// TIA Portal V20 export
FUNCTION_BLOCK "Sequence_1_SepaUnwinderTop"   // FB202, LAD
AUTHOR : ERsystem_FA2_DH. Kim
// stored: IsIECCheckEnabled true, MemoryReserve 100, Namespace Unit1.Em0, SetENOAutomatically false
   VAR
      statSelectedJobNumber { ExternalWritable := 'False'} : DInt;   // Evaluated Job Number
      instSequenceLADStatus { ExternalWritable := 'False'} : "LAF_StatusLadSequence";
      instSequenceLADControl { ExternalWritable := 'False'} : "LAF_ControlLadSequence";
      statTonTime { ExternalAccessible := 'False'; ExternalVisible := 'False'; ExternalWritable := 'False'} : Array[0..1999] of TON_TIME;
   END_VAR
   VAR CONSTANT
      STEP_IDLE : DInt := 1;
      STEP_IMMEDIATE_STOP : DInt := 9001;   // Step executed when an immediate stop command is triggered for the sequence (i.e. when unit is in state aborting)
      JOB_1_STEP_01 : DInt := 101;
      JOB_1_STEP_10 : DInt := 110;
      JOB_1_STEP_20 : DInt := 120;
      JOB_1_STEP_80 : DInt := 180;
      JOB_1_STEP_81 : DInt := 181;
      JOB_1_STEP_90 : DInt := 190;
      JOB_2_STEP_01 : DInt := 201;
      JOB_2_STEP_80 : DInt := 280;
      JOB_2_STEP_90 : DInt := 290;
      JOB_10_STEP_01 : DInt := 1001;
      JOB_10_STEP_80 : DInt := 1080;
      JOB_10_STEP_90 : DInt := 1090;
      FALSE : Bool := FALSE;
      TRUE : Bool := TRUE;
   END_VAR
   VAR_TEMP   // added for the SCL form of the ladder/FBD networks
      _w1 : Bool;
      _w2 : Bool;
   END_VAR
BEGIN

REGION Network 1: BLOCK INFO HEADER
   // (company) / (C) Copyright (year)
   // ---------------------------------------------------------------------------------
   // Title:                             (Title of this block)
   // Comment/Function: (that is implemented in the block)
   // Library/Family:           (that the source is dedicated to)
   // Author:                        (department / person in charge / contact)
   // Target System:          (test system with FW version)
   // Engineering:              TIA Portal (SW version)
   // Restrictions:               (OB types, etc.)
   // Requirements:           (hardware, technological package, etc.)
   // ---------------------------------------------------------------------------------
   // Change log table:
   // Version          | Date             | Signature      | Expert in charge  | Changes applied ------------------------|----------------------|-------------------------|--------------------------------|-----------------------
   // 001.000.000 | yyyy-mm-dd | 0x00000000 | (name of expert) | First released version
END_REGION

REGION Network 2: DESCRIPTION
   // This is a template block provided by the Automation Framework. It can be used to create an own project.
   // The Block Info Header is prepared to put in your own data.
   // Description of the block could be added here and the docu created by Code2Docu.
END_REGION

REGION Network 3: ********************* CONTROL *************************
END_REGION

REGION Network 4: Sequence Control
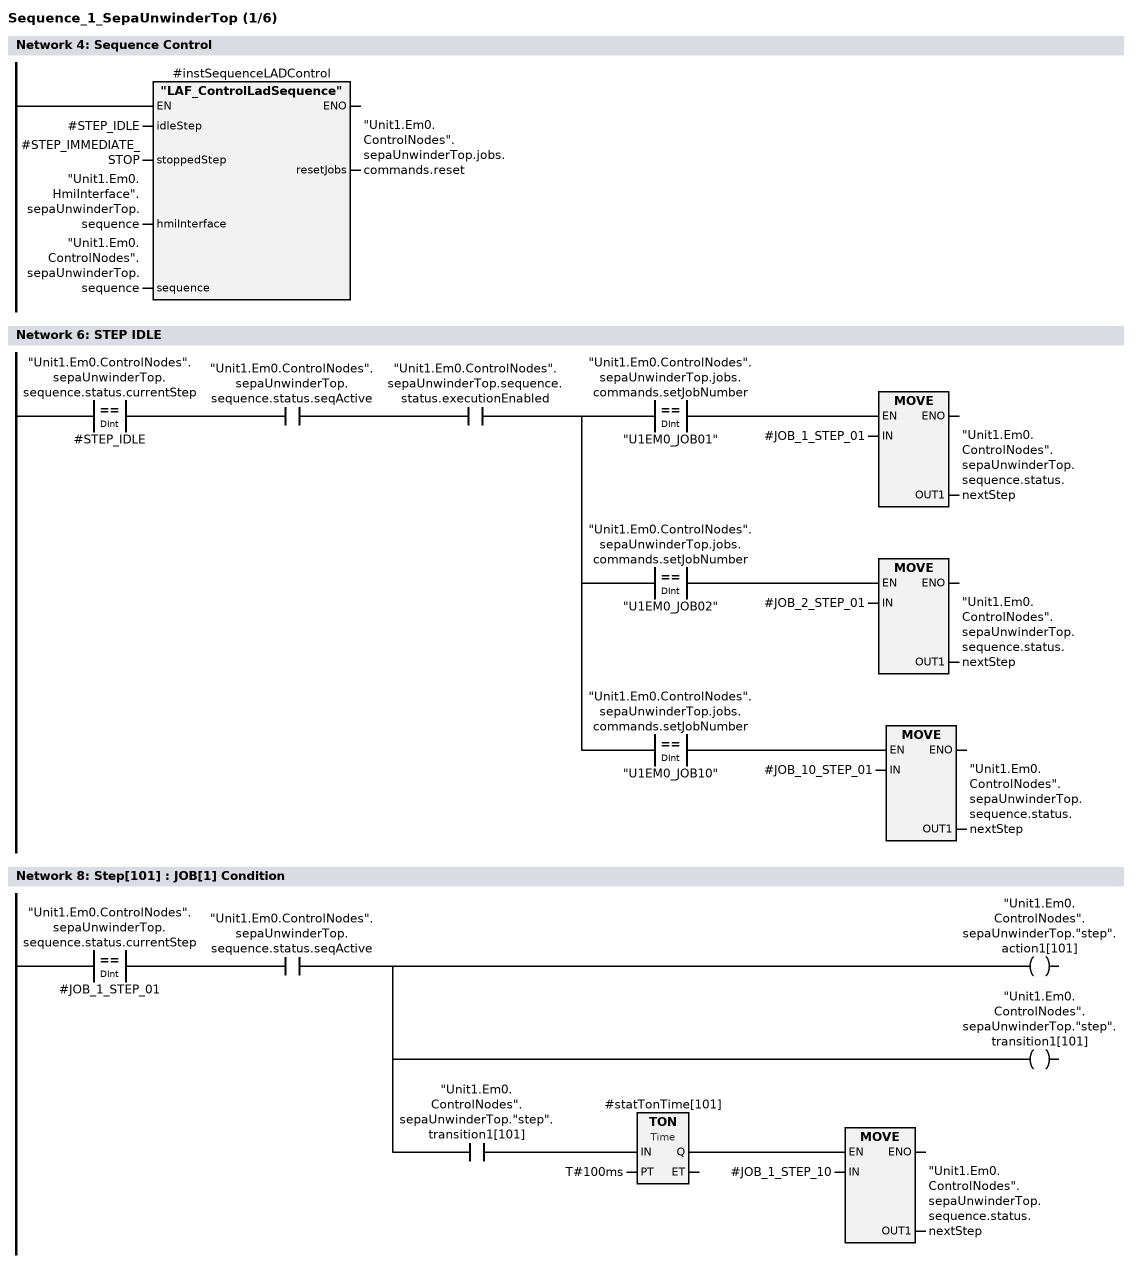
   RUNG wire#powerrail
      #instSequenceLADControl(idleStep := #STEP_IDLE, stoppedStep := #STEP_IMMEDIATE_STOP, hmiInterface := "Unit1.Em0.HmiInterface".sepaUnwinderTop.sequence, sequence := "Unit1.Em0.ControlNodes".sepaUnwinderTop.sequence, resetJobs => "Unit1.Em0.ControlNodes".sepaUnwinderTop.jobs.commands.reset)
   END_RUNG
   // the same network as SCL:
   #instSequenceLADControl(idleStep := #STEP_IDLE,   // "LAF_ControlLadSequence"
                           stoppedStep := #STEP_IMMEDIATE_STOP,
                           hmiInterface := "Unit1.Em0.HmiInterface".sepaUnwinderTop.sequence,
                           sequence := "Unit1.Em0.ControlNodes".sepaUnwinderTop.sequence,
                           resetJobs => "Unit1.Em0.ControlNodes".sepaUnwinderTop.jobs.commands.reset);
END_REGION

REGION Network 5: *************** JOB SELECT **************************
END_REGION

REGION Network 6: STEP IDLE
   RUNG wire#powerrail
      { S7_Templates := "SrcType := DInt" } EQ_Contact(in1 := "Unit1.Em0.ControlNodes".sepaUnwinderTop.sequence.status.currentStep, in2 := #STEP_IDLE)
      Contact( "Unit1.Em0.ControlNodes".sepaUnwinderTop.sequence.status.seqActive )
      Contact( "Unit1.Em0.ControlNodes".sepaUnwinderTop.sequence.status.executionEnabled )
      wire#w1
      { S7_Templates := "SrcType := DInt" } EQ_Contact(in1 := "Unit1.Em0.ControlNodes".sepaUnwinderTop.jobs.commands.setJobNumber, in2 := "U1EM0_JOB01")
      Move(in := #JOB_1_STEP_01, out1 => "Unit1.Em0.ControlNodes".sepaUnwinderTop.sequence.status.nextStep)
   END_RUNG
   RUNG wire#w1
      { S7_Templates := "SrcType := DInt" } EQ_Contact(in1 := "Unit1.Em0.ControlNodes".sepaUnwinderTop.jobs.commands.setJobNumber, in2 := "U1EM0_JOB02")
      Move(in := #JOB_2_STEP_01, out1 => "Unit1.Em0.ControlNodes".sepaUnwinderTop.sequence.status.nextStep)
   END_RUNG
   RUNG wire#w1
      { S7_Templates := "SrcType := DInt" } EQ_Contact(in1 := "Unit1.Em0.ControlNodes".sepaUnwinderTop.jobs.commands.setJobNumber, in2 := "U1EM0_JOB10")
      Move(in := #JOB_10_STEP_01, out1 => "Unit1.Em0.ControlNodes".sepaUnwinderTop.sequence.status.nextStep)
   END_RUNG
   // the same network as SCL:
   #_w1 := ("Unit1.Em0.ControlNodes".sepaUnwinderTop.sequence.status.currentStep = #STEP_IDLE) AND "Unit1.Em0.ControlNodes".sepaUnwinderTop.sequence.status.seqActive AND "Unit1.Em0.ControlNodes".sepaUnwinderTop.sequence.status.executionEnabled;
   IF #_w1 AND ("Unit1.Em0.ControlNodes".sepaUnwinderTop.jobs.commands.setJobNumber = "U1EM0_JOB01") THEN
       "Unit1.Em0.ControlNodes".sepaUnwinderTop.sequence.status.nextStep := #JOB_1_STEP_01;
   END_IF;
   IF #_w1 AND ("Unit1.Em0.ControlNodes".sepaUnwinderTop.jobs.commands.setJobNumber = "U1EM0_JOB02") THEN
       "Unit1.Em0.ControlNodes".sepaUnwinderTop.sequence.status.nextStep := #JOB_2_STEP_01;
   END_IF;
   IF #_w1 AND ("Unit1.Em0.ControlNodes".sepaUnwinderTop.jobs.commands.setJobNumber = "U1EM0_JOB10") THEN
       "Unit1.Em0.ControlNodes".sepaUnwinderTop.sequence.status.nextStep := #JOB_10_STEP_01;
   END_IF;
END_REGION

REGION Network 7: *************** JOB[1] EM HOMING ************************
END_REGION

REGION Network 8: Step[101] : JOB[1] Condition
   RUNG wire#powerrail
      { S7_Templates := "SrcType := DInt" } EQ_Contact(in1 := "Unit1.Em0.ControlNodes".sepaUnwinderTop.sequence.status.currentStep, in2 := #JOB_1_STEP_01)
      Contact( "Unit1.Em0.ControlNodes".sepaUnwinderTop.sequence.status.seqActive )
      wire#w1
      Coil( "Unit1.Em0.ControlNodes".sepaUnwinderTop."step".action1[101] )
   END_RUNG
   RUNG wire#w1
      Coil( "Unit1.Em0.ControlNodes".sepaUnwinderTop."step".transition1[101] )
   END_RUNG
   RUNG wire#w1
      Contact( "Unit1.Em0.ControlNodes".sepaUnwinderTop."step".transition1[101] )
      { S7_Templates := "time_type := Time" } #statTonTime[101].TON(pt := T#100ms, et =>)
      Move(in := #JOB_1_STEP_10, out1 => "Unit1.Em0.ControlNodes".sepaUnwinderTop.sequence.status.nextStep)
   END_RUNG
   // the same network as SCL:
   "Unit1.Em0.ControlNodes".sepaUnwinderTop."step".action1[101] := ("Unit1.Em0.ControlNodes".sepaUnwinderTop.sequence.status.currentStep = #JOB_1_STEP_01) AND "Unit1.Em0.ControlNodes".sepaUnwinderTop.sequence.status.seqActive;
   "Unit1.Em0.ControlNodes".sepaUnwinderTop."step".transition1[101] := ("Unit1.Em0.ControlNodes".sepaUnwinderTop.sequence.status.currentStep = #JOB_1_STEP_01) AND "Unit1.Em0.ControlNodes".sepaUnwinderTop.sequence.status.seqActive;
   #statTonTime[101].TON(IN := ("Unit1.Em0.ControlNodes".sepaUnwinderTop.sequence.status.currentStep = #JOB_1_STEP_01) AND "Unit1.Em0.ControlNodes".sepaUnwinderTop.sequence.status.seqActive AND "Unit1.Em0.ControlNodes".sepaUnwinderTop."step".transition1[101],
                         PT := T#100ms);
   IF #statTonTime[101].Q THEN
       "Unit1.Em0.ControlNodes".sepaUnwinderTop.sequence.status.nextStep := #JOB_1_STEP_10;
   END_IF;
END_REGION

REGION Network 9: Step[110] : Air Shaft On
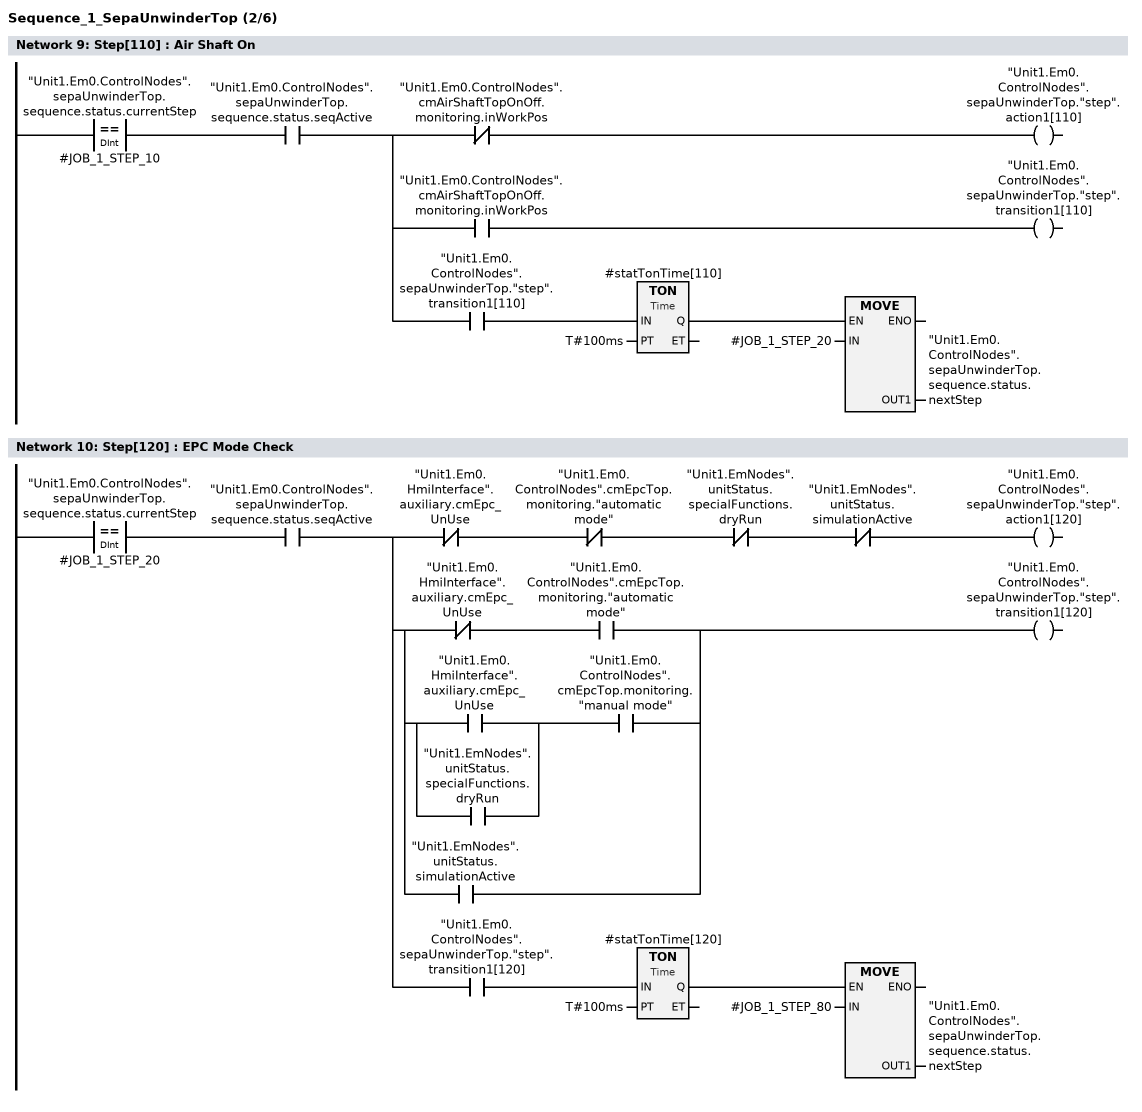
   RUNG wire#powerrail
      { S7_Templates := "SrcType := DInt" } EQ_Contact(in1 := "Unit1.Em0.ControlNodes".sepaUnwinderTop.sequence.status.currentStep, in2 := #JOB_1_STEP_10)
      Contact( "Unit1.Em0.ControlNodes".sepaUnwinderTop.sequence.status.seqActive )
      wire#w1
      I_Contact( "Unit1.Em0.ControlNodes".cmAirShaftTopOnOff.monitoring.inWorkPos )
      Coil( "Unit1.Em0.ControlNodes".sepaUnwinderTop."step".action1[110] )
   END_RUNG
   RUNG wire#w1
      Contact( "Unit1.Em0.ControlNodes".cmAirShaftTopOnOff.monitoring.inWorkPos )
      Coil( "Unit1.Em0.ControlNodes".sepaUnwinderTop."step".transition1[110] )
   END_RUNG
   RUNG wire#w1
      Contact( "Unit1.Em0.ControlNodes".sepaUnwinderTop."step".transition1[110] )
      { S7_Templates := "time_type := Time" } #statTonTime[110].TON(pt := T#100ms, et =>)
      Move(in := #JOB_1_STEP_20, out1 => "Unit1.Em0.ControlNodes".sepaUnwinderTop.sequence.status.nextStep)
   END_RUNG
   // the same network as SCL:
   #_w1 := ("Unit1.Em0.ControlNodes".sepaUnwinderTop.sequence.status.currentStep = #JOB_1_STEP_10) AND "Unit1.Em0.ControlNodes".sepaUnwinderTop.sequence.status.seqActive;
   "Unit1.Em0.ControlNodes".sepaUnwinderTop."step".action1[110] := #_w1 AND NOT "Unit1.Em0.ControlNodes".cmAirShaftTopOnOff.monitoring.inWorkPos;
   "Unit1.Em0.ControlNodes".sepaUnwinderTop."step".transition1[110] := #_w1 AND "Unit1.Em0.ControlNodes".cmAirShaftTopOnOff.monitoring.inWorkPos;
   #statTonTime[110].TON(IN := #_w1 AND "Unit1.Em0.ControlNodes".sepaUnwinderTop."step".transition1[110],
                         PT := T#100ms);
   IF #statTonTime[110].Q THEN
       "Unit1.Em0.ControlNodes".sepaUnwinderTop.sequence.status.nextStep := #JOB_1_STEP_20;
   END_IF;
END_REGION

REGION Network 10: Step[120] : EPC Mode Check
   RUNG wire#powerrail
      { S7_Templates := "SrcType := DInt" } EQ_Contact(in1 := "Unit1.Em0.ControlNodes".sepaUnwinderTop.sequence.status.currentStep, in2 := #JOB_1_STEP_20)
      Contact( "Unit1.Em0.ControlNodes".sepaUnwinderTop.sequence.status.seqActive )
      wire#w1
      I_Contact( "Unit1.Em0.HmiInterface".auxiliary.cmEpc_UnUse )
      I_Contact( "Unit1.Em0.ControlNodes".cmEpcTop.monitoring."automatic mode" )
      I_Contact( "Unit1.EmNodes".unitStatus.specialFunctions.dryRun )
      I_Contact( "Unit1.EmNodes".unitStatus.simulationActive )
      Coil( "Unit1.Em0.ControlNodes".sepaUnwinderTop."step".action1[120] )
   END_RUNG
   RUNG wire#w1
      I_Contact( "Unit1.Em0.HmiInterface".auxiliary.cmEpc_UnUse )
      Contact( "Unit1.Em0.ControlNodes".cmEpcTop.monitoring."automatic mode" )
      wire#w2
      Coil( "Unit1.Em0.ControlNodes".sepaUnwinderTop."step".transition1[120] )
   END_RUNG
   RUNG wire#w1
      Contact( "Unit1.Em0.HmiInterface".auxiliary.cmEpc_UnUse )
      wire#w3
      Contact( "Unit1.Em0.ControlNodes".cmEpcTop.monitoring."manual mode" )
   END_RUNG wire#w2
   RUNG wire#w1
      Contact( "Unit1.EmNodes".unitStatus.specialFunctions.dryRun )
   END_RUNG wire#w3
   RUNG wire#w1
      Contact( "Unit1.EmNodes".unitStatus.simulationActive )
   END_RUNG wire#w2
   RUNG wire#w1
      Contact( "Unit1.Em0.ControlNodes".sepaUnwinderTop."step".transition1[120] )
      { S7_Templates := "time_type := Time" } #statTonTime[120].TON(pt := T#100ms, et =>)
      Move(in := #JOB_1_STEP_80, out1 => "Unit1.Em0.ControlNodes".sepaUnwinderTop.sequence.status.nextStep)
   END_RUNG
   // the same network as SCL:
   #_w1 := ("Unit1.Em0.ControlNodes".sepaUnwinderTop.sequence.status.currentStep = #JOB_1_STEP_20) AND "Unit1.Em0.ControlNodes".sepaUnwinderTop.sequence.status.seqActive;
   "Unit1.Em0.ControlNodes".sepaUnwinderTop."step".action1[120] := #_w1 AND NOT "Unit1.Em0.HmiInterface".auxiliary.cmEpc_UnUse AND NOT "Unit1.Em0.ControlNodes".cmEpcTop.monitoring."automatic mode" AND NOT "Unit1.EmNodes".unitStatus.specialFunctions.dryRun AND NOT "Unit1.EmNodes".unitStatus.simulationActive;
   "Unit1.Em0.ControlNodes".sepaUnwinderTop."step".transition1[120] := #_w1 AND ((NOT "Unit1.Em0.HmiInterface".auxiliary.cmEpc_UnUse AND "Unit1.Em0.ControlNodes".cmEpcTop.monitoring."automatic mode") OR (("Unit1.Em0.HmiInterface".auxiliary.cmEpc_UnUse OR "Unit1.EmNodes".unitStatus.specialFunctions.dryRun) AND "Unit1.Em0.ControlNodes".cmEpcTop.monitoring."manual mode") OR "Unit1.EmNodes".unitStatus.simulationActive);
   #statTonTime[120].TON(IN := #_w1 AND "Unit1.Em0.ControlNodes".sepaUnwinderTop."step".transition1[120],
                         PT := T#100ms);
   IF #statTonTime[120].Q THEN
       "Unit1.Em0.ControlNodes".sepaUnwinderTop.sequence.status.nextStep := #JOB_1_STEP_80;
   END_IF;
END_REGION

REGION Network 11: Step[180] : Unwinder B-Axis Jog Commands
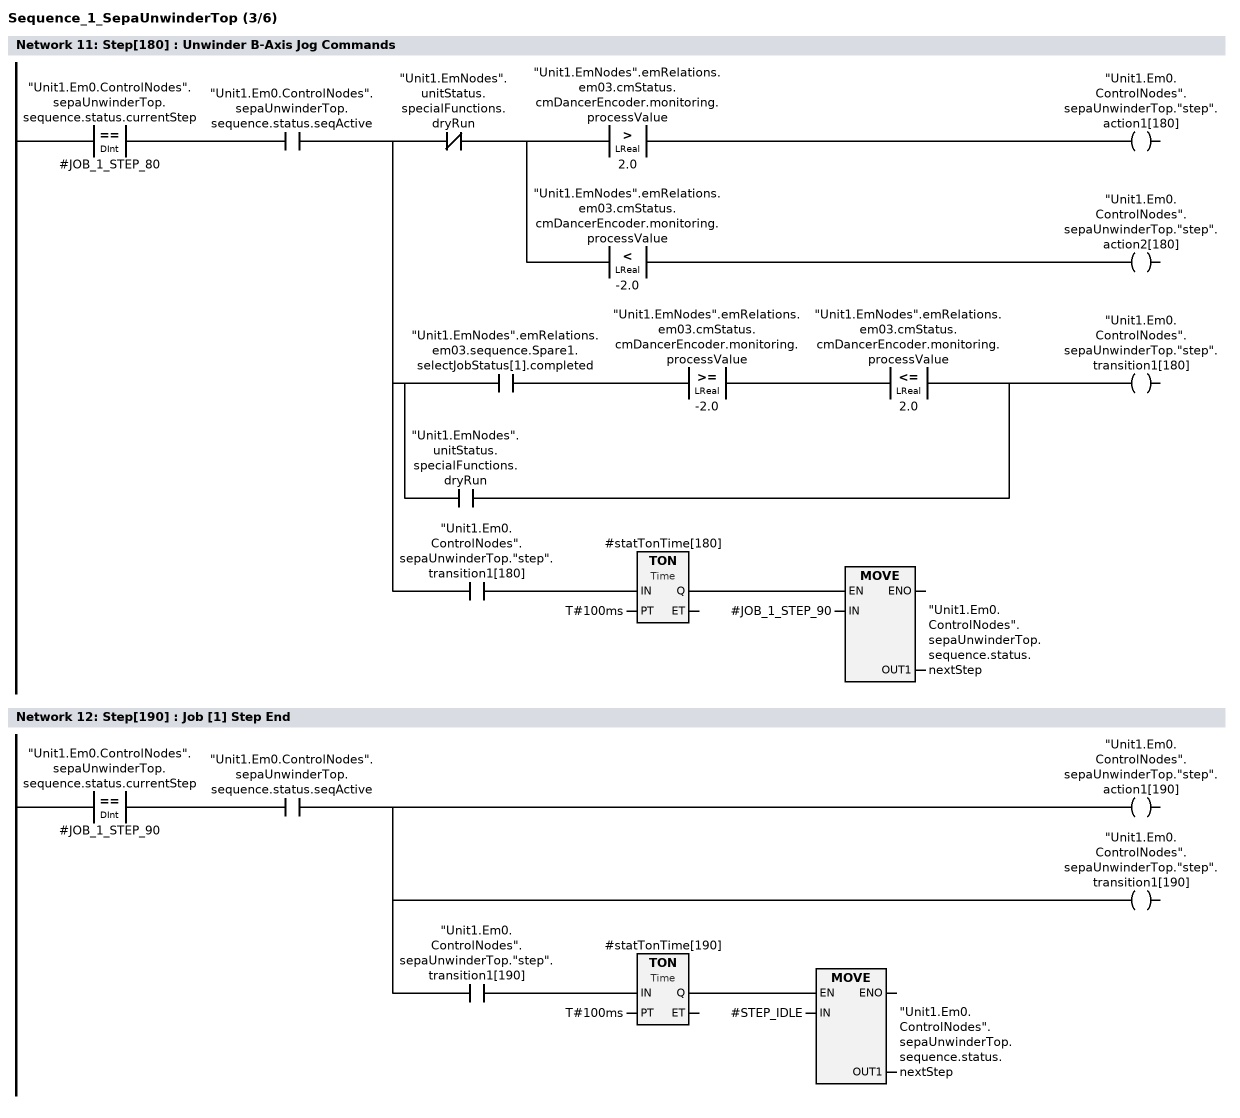
   RUNG wire#powerrail
      { S7_Templates := "SrcType := DInt" } EQ_Contact(in1 := "Unit1.Em0.ControlNodes".sepaUnwinderTop.sequence.status.currentStep, in2 := #JOB_1_STEP_80)
      Contact( "Unit1.Em0.ControlNodes".sepaUnwinderTop.sequence.status.seqActive )
      wire#w1
      I_Contact( "Unit1.EmNodes".unitStatus.specialFunctions.dryRun )
      wire#w2
      { S7_Templates := "SrcType := LReal" } GT_Contact(in1 := "Unit1.EmNodes".emRelations.em03.cmStatus.cmDancerEncoder.monitoring.processValue, in2 := 2.0)
      Coil( "Unit1.Em0.ControlNodes".sepaUnwinderTop."step".action1[180] )
   END_RUNG
   RUNG wire#w2
      { S7_Templates := "SrcType := LReal" } LT_Contact(in1 := "Unit1.EmNodes".emRelations.em03.cmStatus.cmDancerEncoder.monitoring.processValue, in2 := -2.0)
      Coil( "Unit1.Em0.ControlNodes".sepaUnwinderTop."step".action2[180] )
   END_RUNG
   RUNG wire#w1
      Contact( "Unit1.EmNodes".emRelations.em03.sequence.Spare1.selectJobStatus[1].completed )
      { S7_Templates := "SrcType := LReal" } GE_Contact(in1 := "Unit1.EmNodes".emRelations.em03.cmStatus.cmDancerEncoder.monitoring.processValue, in2 := -2.0)
      { S7_Templates := "SrcType := LReal" } LE_Contact(in1 := "Unit1.EmNodes".emRelations.em03.cmStatus.cmDancerEncoder.monitoring.processValue, in2 := 2.0)
      wire#w3
      Coil( "Unit1.Em0.ControlNodes".sepaUnwinderTop."step".transition1[180] )
   END_RUNG
   RUNG wire#w1
      Contact( "Unit1.EmNodes".unitStatus.specialFunctions.dryRun )
   END_RUNG wire#w3
   RUNG wire#w1
      Contact( "Unit1.Em0.ControlNodes".sepaUnwinderTop."step".transition1[180] )
      { S7_Templates := "time_type := Time" } #statTonTime[180].TON(pt := T#100ms, et =>)
      Move(in := #JOB_1_STEP_90, out1 => "Unit1.Em0.ControlNodes".sepaUnwinderTop.sequence.status.nextStep)
   END_RUNG
   // the same network as SCL:
   #_w1 := ("Unit1.Em0.ControlNodes".sepaUnwinderTop.sequence.status.currentStep = #JOB_1_STEP_80) AND "Unit1.Em0.ControlNodes".sepaUnwinderTop.sequence.status.seqActive;
   #_w2 := #_w1 AND NOT "Unit1.EmNodes".unitStatus.specialFunctions.dryRun;
   "Unit1.Em0.ControlNodes".sepaUnwinderTop."step".action1[180] := #_w2 AND ("Unit1.EmNodes".emRelations.em03.cmStatus.cmDancerEncoder.monitoring.processValue > 2.0);
   "Unit1.Em0.ControlNodes".sepaUnwinderTop."step".action2[180] := #_w2 AND ("Unit1.EmNodes".emRelations.em03.cmStatus.cmDancerEncoder.monitoring.processValue < (-2.0));
   "Unit1.Em0.ControlNodes".sepaUnwinderTop."step".transition1[180] := #_w1 AND (("Unit1.EmNodes".emRelations.em03.sequence.Spare1.selectJobStatus[1].completed AND ("Unit1.EmNodes".emRelations.em03.cmStatus.cmDancerEncoder.monitoring.processValue >= (-2.0)) AND ("Unit1.EmNodes".emRelations.em03.cmStatus.cmDancerEncoder.monitoring.processValue <= 2.0)) OR "Unit1.EmNodes".unitStatus.specialFunctions.dryRun);
   #statTonTime[180].TON(IN := #_w1 AND "Unit1.Em0.ControlNodes".sepaUnwinderTop."step".transition1[180],
                         PT := T#100ms);
   IF #statTonTime[180].Q THEN
       "Unit1.Em0.ControlNodes".sepaUnwinderTop.sequence.status.nextStep := #JOB_1_STEP_90;
   END_IF;
END_REGION

REGION Network 12: Step[190] : Job [1] Step End
   RUNG wire#powerrail
      { S7_Templates := "SrcType := DInt" } EQ_Contact(in1 := "Unit1.Em0.ControlNodes".sepaUnwinderTop.sequence.status.currentStep, in2 := #JOB_1_STEP_90)
      Contact( "Unit1.Em0.ControlNodes".sepaUnwinderTop.sequence.status.seqActive )
      wire#w1
      Coil( "Unit1.Em0.ControlNodes".sepaUnwinderTop."step".action1[190] )
   END_RUNG
   RUNG wire#w1
      Coil( "Unit1.Em0.ControlNodes".sepaUnwinderTop."step".transition1[190] )
   END_RUNG
   RUNG wire#w1
      Contact( "Unit1.Em0.ControlNodes".sepaUnwinderTop."step".transition1[190] )
      { S7_Templates := "time_type := Time" } #statTonTime[190].TON(pt := T#100ms, et =>)
      Move(in := #STEP_IDLE, out1 => "Unit1.Em0.ControlNodes".sepaUnwinderTop.sequence.status.nextStep)
   END_RUNG
   // the same network as SCL:
   "Unit1.Em0.ControlNodes".sepaUnwinderTop."step".action1[190] := ("Unit1.Em0.ControlNodes".sepaUnwinderTop.sequence.status.currentStep = #JOB_1_STEP_90) AND "Unit1.Em0.ControlNodes".sepaUnwinderTop.sequence.status.seqActive;
   "Unit1.Em0.ControlNodes".sepaUnwinderTop."step".transition1[190] := ("Unit1.Em0.ControlNodes".sepaUnwinderTop.sequence.status.currentStep = #JOB_1_STEP_90) AND "Unit1.Em0.ControlNodes".sepaUnwinderTop.sequence.status.seqActive;
   #statTonTime[190].TON(IN := ("Unit1.Em0.ControlNodes".sepaUnwinderTop.sequence.status.currentStep = #JOB_1_STEP_90) AND "Unit1.Em0.ControlNodes".sepaUnwinderTop.sequence.status.seqActive AND "Unit1.Em0.ControlNodes".sepaUnwinderTop."step".transition1[190],
                         PT := T#100ms);
   IF #statTonTime[190].Q THEN
       "Unit1.Em0.ControlNodes".sepaUnwinderTop.sequence.status.nextStep := #STEP_IDLE;
   END_IF;
END_REGION

REGION Network 13: ******************** JOB[2] Motion ********************
END_REGION

REGION Network 14: Step[201] : JOB[2] Condition
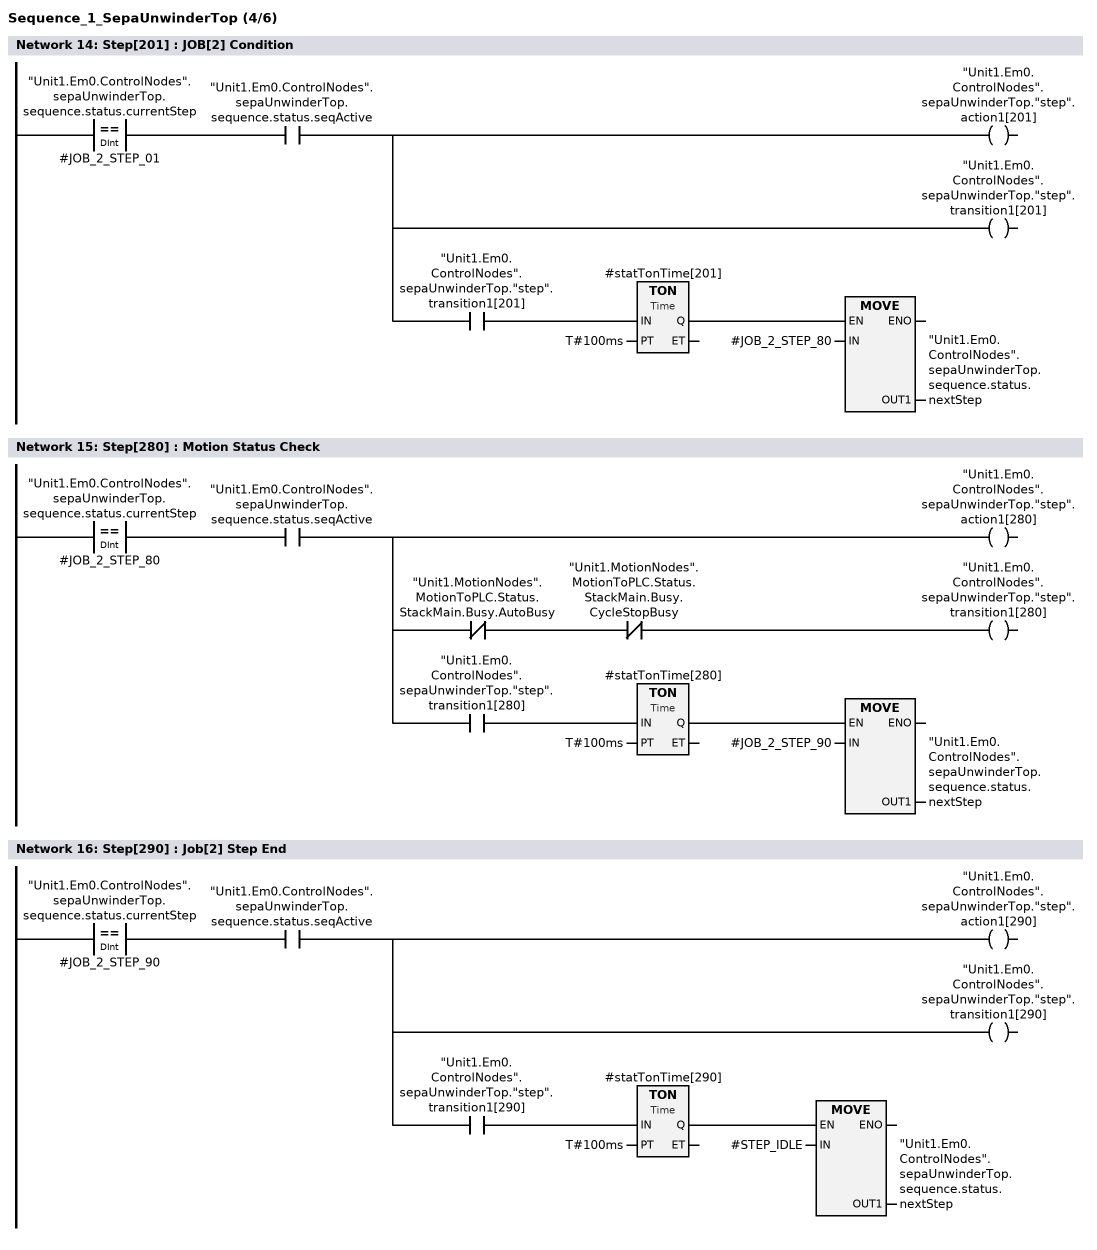
   RUNG wire#powerrail
      { S7_Templates := "SrcType := DInt" } EQ_Contact(in1 := "Unit1.Em0.ControlNodes".sepaUnwinderTop.sequence.status.currentStep, in2 := #JOB_2_STEP_01)
      Contact( "Unit1.Em0.ControlNodes".sepaUnwinderTop.sequence.status.seqActive )
      wire#w1
      Coil( "Unit1.Em0.ControlNodes".sepaUnwinderTop."step".action1[201] )
   END_RUNG
   RUNG wire#w1
      Coil( "Unit1.Em0.ControlNodes".sepaUnwinderTop."step".transition1[201] )
   END_RUNG
   RUNG wire#w1
      Contact( "Unit1.Em0.ControlNodes".sepaUnwinderTop."step".transition1[201] )
      { S7_Templates := "time_type := Time" } #statTonTime[201].TON(pt := T#100ms, et =>)
      Move(in := #JOB_2_STEP_80, out1 => "Unit1.Em0.ControlNodes".sepaUnwinderTop.sequence.status.nextStep)
   END_RUNG
   // the same network as SCL:
   "Unit1.Em0.ControlNodes".sepaUnwinderTop."step".action1[201] := ("Unit1.Em0.ControlNodes".sepaUnwinderTop.sequence.status.currentStep = #JOB_2_STEP_01) AND "Unit1.Em0.ControlNodes".sepaUnwinderTop.sequence.status.seqActive;
   "Unit1.Em0.ControlNodes".sepaUnwinderTop."step".transition1[201] := ("Unit1.Em0.ControlNodes".sepaUnwinderTop.sequence.status.currentStep = #JOB_2_STEP_01) AND "Unit1.Em0.ControlNodes".sepaUnwinderTop.sequence.status.seqActive;
   #statTonTime[201].TON(IN := ("Unit1.Em0.ControlNodes".sepaUnwinderTop.sequence.status.currentStep = #JOB_2_STEP_01) AND "Unit1.Em0.ControlNodes".sepaUnwinderTop.sequence.status.seqActive AND "Unit1.Em0.ControlNodes".sepaUnwinderTop."step".transition1[201],
                         PT := T#100ms);
   IF #statTonTime[201].Q THEN
       "Unit1.Em0.ControlNodes".sepaUnwinderTop.sequence.status.nextStep := #JOB_2_STEP_80;
   END_IF;
END_REGION

REGION Network 15: Step[280] : Motion Status Check
   RUNG wire#powerrail
      { S7_Templates := "SrcType := DInt" } EQ_Contact(in1 := "Unit1.Em0.ControlNodes".sepaUnwinderTop.sequence.status.currentStep, in2 := #JOB_2_STEP_80)
      Contact( "Unit1.Em0.ControlNodes".sepaUnwinderTop.sequence.status.seqActive )
      wire#w1
      Coil( "Unit1.Em0.ControlNodes".sepaUnwinderTop."step".action1[280] )
   END_RUNG
   RUNG wire#w1
      I_Contact( "Unit1.MotionNodes".MotionToPLC.Status.StackMain.Busy.AutoBusy )
      I_Contact( "Unit1.MotionNodes".MotionToPLC.Status.StackMain.Busy.CycleStopBusy )
      Coil( "Unit1.Em0.ControlNodes".sepaUnwinderTop."step".transition1[280] )
   END_RUNG
   RUNG wire#w1
      Contact( "Unit1.Em0.ControlNodes".sepaUnwinderTop."step".transition1[280] )
      { S7_Templates := "time_type := Time" } #statTonTime[280].TON(pt := T#100ms, et =>)
      Move(in := #JOB_2_STEP_90, out1 => "Unit1.Em0.ControlNodes".sepaUnwinderTop.sequence.status.nextStep)
   END_RUNG
   // the same network as SCL:
   "Unit1.Em0.ControlNodes".sepaUnwinderTop."step".action1[280] := ("Unit1.Em0.ControlNodes".sepaUnwinderTop.sequence.status.currentStep = #JOB_2_STEP_80) AND "Unit1.Em0.ControlNodes".sepaUnwinderTop.sequence.status.seqActive;
   "Unit1.Em0.ControlNodes".sepaUnwinderTop."step".transition1[280] := ("Unit1.Em0.ControlNodes".sepaUnwinderTop.sequence.status.currentStep = #JOB_2_STEP_80) AND "Unit1.Em0.ControlNodes".sepaUnwinderTop.sequence.status.seqActive AND NOT "Unit1.MotionNodes".MotionToPLC.Status.StackMain.Busy.AutoBusy AND NOT "Unit1.MotionNodes".MotionToPLC.Status.StackMain.Busy.CycleStopBusy;
   #statTonTime[280].TON(IN := ("Unit1.Em0.ControlNodes".sepaUnwinderTop.sequence.status.currentStep = #JOB_2_STEP_80) AND "Unit1.Em0.ControlNodes".sepaUnwinderTop.sequence.status.seqActive AND "Unit1.Em0.ControlNodes".sepaUnwinderTop."step".transition1[280],
                         PT := T#100ms);
   IF #statTonTime[280].Q THEN
       "Unit1.Em0.ControlNodes".sepaUnwinderTop.sequence.status.nextStep := #JOB_2_STEP_90;
   END_IF;
END_REGION

REGION Network 16: Step[290] : Job[2] Step End
   RUNG wire#powerrail
      { S7_Templates := "SrcType := DInt" } EQ_Contact(in1 := "Unit1.Em0.ControlNodes".sepaUnwinderTop.sequence.status.currentStep, in2 := #JOB_2_STEP_90)
      Contact( "Unit1.Em0.ControlNodes".sepaUnwinderTop.sequence.status.seqActive )
      wire#w1
      Coil( "Unit1.Em0.ControlNodes".sepaUnwinderTop."step".action1[290] )
   END_RUNG
   RUNG wire#w1
      Coil( "Unit1.Em0.ControlNodes".sepaUnwinderTop."step".transition1[290] )
   END_RUNG
   RUNG wire#w1
      Contact( "Unit1.Em0.ControlNodes".sepaUnwinderTop."step".transition1[290] )
      { S7_Templates := "time_type := Time" } #statTonTime[290].TON(pt := T#100ms, et =>)
      Move(in := #STEP_IDLE, out1 => "Unit1.Em0.ControlNodes".sepaUnwinderTop.sequence.status.nextStep)
   END_RUNG
   // the same network as SCL:
   "Unit1.Em0.ControlNodes".sepaUnwinderTop."step".action1[290] := ("Unit1.Em0.ControlNodes".sepaUnwinderTop.sequence.status.currentStep = #JOB_2_STEP_90) AND "Unit1.Em0.ControlNodes".sepaUnwinderTop.sequence.status.seqActive;
   "Unit1.Em0.ControlNodes".sepaUnwinderTop."step".transition1[290] := ("Unit1.Em0.ControlNodes".sepaUnwinderTop.sequence.status.currentStep = #JOB_2_STEP_90) AND "Unit1.Em0.ControlNodes".sepaUnwinderTop.sequence.status.seqActive;
   #statTonTime[290].TON(IN := ("Unit1.Em0.ControlNodes".sepaUnwinderTop.sequence.status.currentStep = #JOB_2_STEP_90) AND "Unit1.Em0.ControlNodes".sepaUnwinderTop.sequence.status.seqActive AND "Unit1.Em0.ControlNodes".sepaUnwinderTop."step".transition1[290],
                         PT := T#100ms);
   IF #statTonTime[290].Q THEN
       "Unit1.Em0.ControlNodes".sepaUnwinderTop.sequence.status.nextStep := #STEP_IDLE;
   END_IF;
END_REGION

REGION Network 17: *************** JOB[10] REWINDING[AUTO SPLICING] ************************
END_REGION

REGION Network 18: Step[1001] : JOB[10] Condition
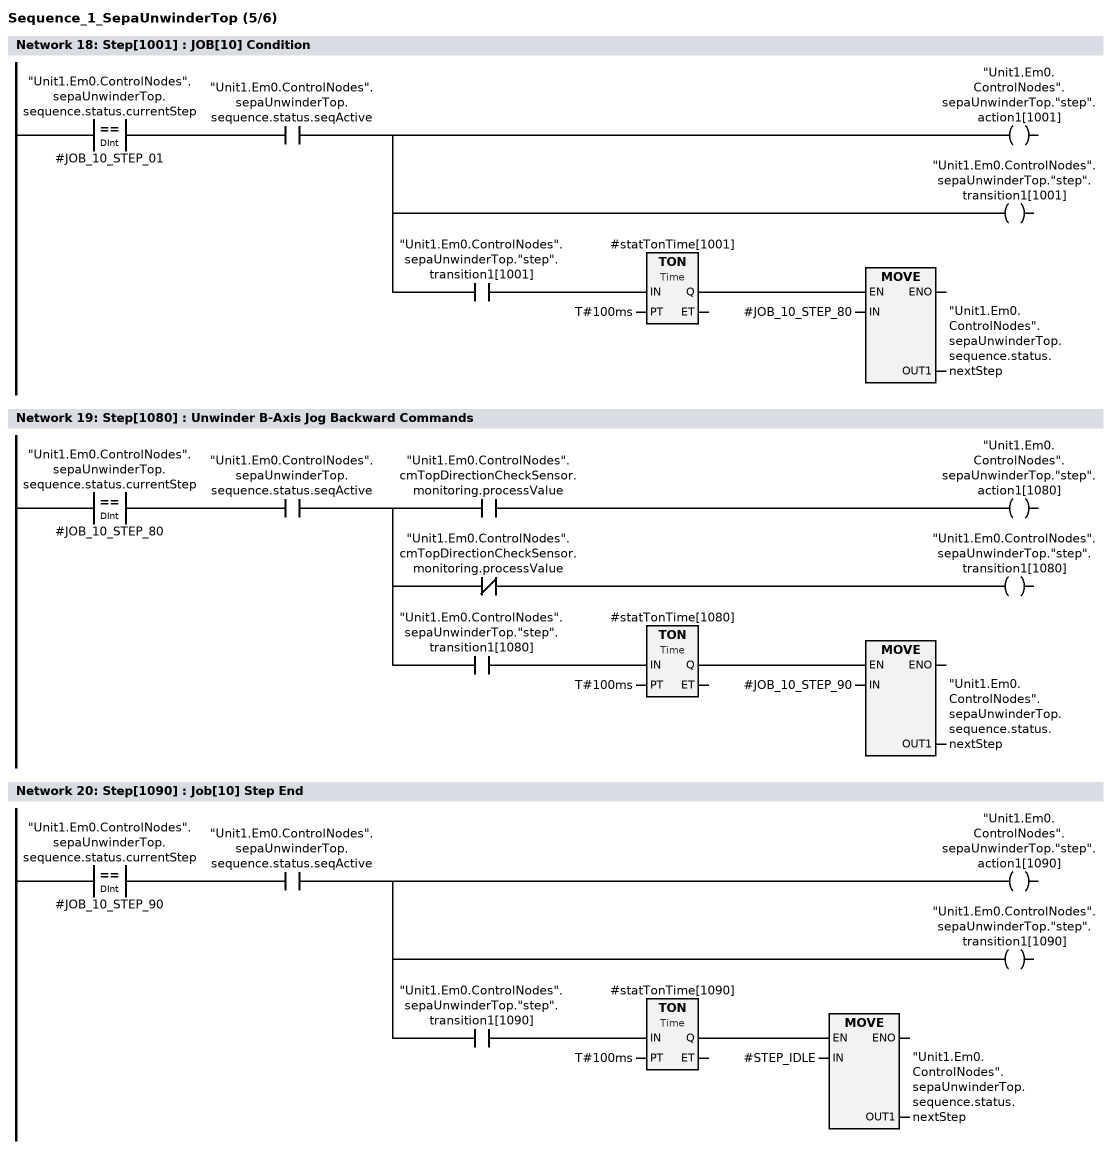
   RUNG wire#powerrail
      { S7_Templates := "SrcType := DInt" } EQ_Contact(in1 := "Unit1.Em0.ControlNodes".sepaUnwinderTop.sequence.status.currentStep, in2 := #JOB_10_STEP_01)
      Contact( "Unit1.Em0.ControlNodes".sepaUnwinderTop.sequence.status.seqActive )
      wire#w1
      Coil( "Unit1.Em0.ControlNodes".sepaUnwinderTop."step".action1[1001] )
   END_RUNG
   RUNG wire#w1
      Coil( "Unit1.Em0.ControlNodes".sepaUnwinderTop."step".transition1[1001] )
   END_RUNG
   RUNG wire#w1
      Contact( "Unit1.Em0.ControlNodes".sepaUnwinderTop."step".transition1[1001] )
      { S7_Templates := "time_type := Time" } #statTonTime[1001].TON(pt := T#100ms, et =>)
      Move(in := #JOB_10_STEP_80, out1 => "Unit1.Em0.ControlNodes".sepaUnwinderTop.sequence.status.nextStep)
   END_RUNG
   // the same network as SCL:
   "Unit1.Em0.ControlNodes".sepaUnwinderTop."step".action1[1001] := ("Unit1.Em0.ControlNodes".sepaUnwinderTop.sequence.status.currentStep = #JOB_10_STEP_01) AND "Unit1.Em0.ControlNodes".sepaUnwinderTop.sequence.status.seqActive;
   "Unit1.Em0.ControlNodes".sepaUnwinderTop."step".transition1[1001] := ("Unit1.Em0.ControlNodes".sepaUnwinderTop.sequence.status.currentStep = #JOB_10_STEP_01) AND "Unit1.Em0.ControlNodes".sepaUnwinderTop.sequence.status.seqActive;
   #statTonTime[1001].TON(IN := ("Unit1.Em0.ControlNodes".sepaUnwinderTop.sequence.status.currentStep = #JOB_10_STEP_01) AND "Unit1.Em0.ControlNodes".sepaUnwinderTop.sequence.status.seqActive AND "Unit1.Em0.ControlNodes".sepaUnwinderTop."step".transition1[1001],
                          PT := T#100ms);
   IF #statTonTime[1001].Q THEN
       "Unit1.Em0.ControlNodes".sepaUnwinderTop.sequence.status.nextStep := #JOB_10_STEP_80;
   END_IF;
END_REGION

REGION Network 19: Step[1080] : Unwinder B-Axis Jog Backward Commands
   RUNG wire#powerrail
      { S7_Templates := "SrcType := DInt" } EQ_Contact(in1 := "Unit1.Em0.ControlNodes".sepaUnwinderTop.sequence.status.currentStep, in2 := #JOB_10_STEP_80)
      Contact( "Unit1.Em0.ControlNodes".sepaUnwinderTop.sequence.status.seqActive )
      wire#w1
      Contact( "Unit1.Em0.ControlNodes".cmTopDirectionCheckSensor.monitoring.processValue )
      Coil( "Unit1.Em0.ControlNodes".sepaUnwinderTop."step".action1[1080] )
   END_RUNG
   RUNG wire#w1
      I_Contact( "Unit1.Em0.ControlNodes".cmTopDirectionCheckSensor.monitoring.processValue )
      Coil( "Unit1.Em0.ControlNodes".sepaUnwinderTop."step".transition1[1080] )
   END_RUNG
   RUNG wire#w1
      Contact( "Unit1.Em0.ControlNodes".sepaUnwinderTop."step".transition1[1080] )
      { S7_Templates := "time_type := Time" } #statTonTime[1080].TON(pt := T#100ms, et =>)
      Move(in := #JOB_10_STEP_90, out1 => "Unit1.Em0.ControlNodes".sepaUnwinderTop.sequence.status.nextStep)
   END_RUNG
   // the same network as SCL:
   #_w1 := ("Unit1.Em0.ControlNodes".sepaUnwinderTop.sequence.status.currentStep = #JOB_10_STEP_80) AND "Unit1.Em0.ControlNodes".sepaUnwinderTop.sequence.status.seqActive;
   "Unit1.Em0.ControlNodes".sepaUnwinderTop."step".action1[1080] := #_w1 AND "Unit1.Em0.ControlNodes".cmTopDirectionCheckSensor.monitoring.processValue;
   "Unit1.Em0.ControlNodes".sepaUnwinderTop."step".transition1[1080] := #_w1 AND NOT "Unit1.Em0.ControlNodes".cmTopDirectionCheckSensor.monitoring.processValue;
   #statTonTime[1080].TON(IN := #_w1 AND "Unit1.Em0.ControlNodes".sepaUnwinderTop."step".transition1[1080],
                          PT := T#100ms);
   IF #statTonTime[1080].Q THEN
       "Unit1.Em0.ControlNodes".sepaUnwinderTop.sequence.status.nextStep := #JOB_10_STEP_90;
   END_IF;
END_REGION

REGION Network 20: Step[1090] : Job[10] Step End
   RUNG wire#powerrail
      { S7_Templates := "SrcType := DInt" } EQ_Contact(in1 := "Unit1.Em0.ControlNodes".sepaUnwinderTop.sequence.status.currentStep, in2 := #JOB_10_STEP_90)
      Contact( "Unit1.Em0.ControlNodes".sepaUnwinderTop.sequence.status.seqActive )
      wire#w1
      Coil( "Unit1.Em0.ControlNodes".sepaUnwinderTop."step".action1[1090] )
   END_RUNG
   RUNG wire#w1
      Coil( "Unit1.Em0.ControlNodes".sepaUnwinderTop."step".transition1[1090] )
   END_RUNG
   RUNG wire#w1
      Contact( "Unit1.Em0.ControlNodes".sepaUnwinderTop."step".transition1[1090] )
      { S7_Templates := "time_type := Time" } #statTonTime[1090].TON(pt := T#100ms, et =>)
      Move(in := #STEP_IDLE, out1 => "Unit1.Em0.ControlNodes".sepaUnwinderTop.sequence.status.nextStep)
   END_RUNG
   // the same network as SCL:
   "Unit1.Em0.ControlNodes".sepaUnwinderTop."step".action1[1090] := ("Unit1.Em0.ControlNodes".sepaUnwinderTop.sequence.status.currentStep = #JOB_10_STEP_90) AND "Unit1.Em0.ControlNodes".sepaUnwinderTop.sequence.status.seqActive;
   "Unit1.Em0.ControlNodes".sepaUnwinderTop."step".transition1[1090] := ("Unit1.Em0.ControlNodes".sepaUnwinderTop.sequence.status.currentStep = #JOB_10_STEP_90) AND "Unit1.Em0.ControlNodes".sepaUnwinderTop.sequence.status.seqActive;
   #statTonTime[1090].TON(IN := ("Unit1.Em0.ControlNodes".sepaUnwinderTop.sequence.status.currentStep = #JOB_10_STEP_90) AND "Unit1.Em0.ControlNodes".sepaUnwinderTop.sequence.status.seqActive AND "Unit1.Em0.ControlNodes".sepaUnwinderTop."step".transition1[1090],
                          PT := T#100ms);
   IF #statTonTime[1090].Q THEN
       "Unit1.Em0.ControlNodes".sepaUnwinderTop.sequence.status.nextStep := #STEP_IDLE;
   END_IF;
END_REGION

REGION Network 21: *************** IMMEDIATE STOP **************************
END_REGION

REGION Network 22: Immediate Stop
END_REGION

REGION Network 23: *************** Status updates **************************
END_REGION

REGION Network 24: Sequence Status
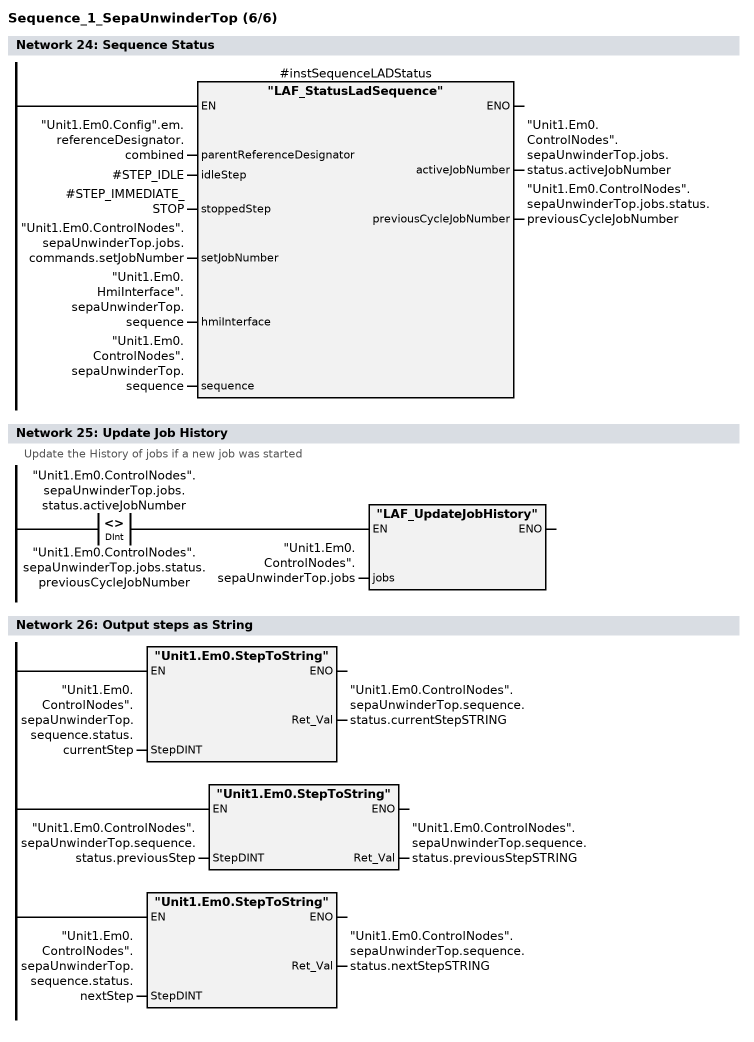
   RUNG wire#powerrail
      #instSequenceLADStatus(parentReferenceDesignator := "Unit1.Em0.Config".em.referenceDesignator.combined, idleStep := #STEP_IDLE, stoppedStep := #STEP_IMMEDIATE_STOP, setJobNumber := "Unit1.Em0.ControlNodes".sepaUnwinderTop.jobs.commands.setJobNumber, hmiInterface := "Unit1.Em0.HmiInterface".sepaUnwinderTop.sequence, sequence := "Unit1.Em0.ControlNodes".sepaUnwinderTop.sequence, activeJobNumber => "Unit1.Em0.ControlNodes".sepaUnwinderTop.jobs.status.activeJobNumber, previousCycleJobNumber => "Unit1.Em0.ControlNodes".sepaUnwinderTop.jobs.status.previousCycleJobNumber)
   END_RUNG
   // the same network as SCL:
   #instSequenceLADStatus(parentReferenceDesignator := "Unit1.Em0.Config".em.referenceDesignator.combined,   // "LAF_StatusLadSequence"
                          idleStep := #STEP_IDLE,
                          stoppedStep := #STEP_IMMEDIATE_STOP,
                          setJobNumber := "Unit1.Em0.ControlNodes".sepaUnwinderTop.jobs.commands.setJobNumber,
                          hmiInterface := "Unit1.Em0.HmiInterface".sepaUnwinderTop.sequence,
                          sequence := "Unit1.Em0.ControlNodes".sepaUnwinderTop.sequence,
                          activeJobNumber => "Unit1.Em0.ControlNodes".sepaUnwinderTop.jobs.status.activeJobNumber,
                          previousCycleJobNumber => "Unit1.Em0.ControlNodes".sepaUnwinderTop.jobs.status.previousCycleJobNumber);
END_REGION

REGION Network 25: Update Job History
   // Update the History of jobs if a new job was started
   RUNG wire#powerrail
      { S7_Templates := "SrcType := DInt" } NE_Contact(in1 := "Unit1.Em0.ControlNodes".sepaUnwinderTop.jobs.status.activeJobNumber, in2 := "Unit1.Em0.ControlNodes".sepaUnwinderTop.jobs.status.previousCycleJobNumber)
      "LAF_UpdateJobHistory"(jobs := "Unit1.Em0.ControlNodes".sepaUnwinderTop.jobs)
   END_RUNG
   // the same network as SCL:
   IF "Unit1.Em0.ControlNodes".sepaUnwinderTop.jobs.status.activeJobNumber <> "Unit1.Em0.ControlNodes".sepaUnwinderTop.jobs.status.previousCycleJobNumber THEN
       "LAF_UpdateJobHistory"(jobs := "Unit1.Em0.ControlNodes".sepaUnwinderTop.jobs);
   END_IF;
END_REGION

REGION Network 26: Output steps as String
   RUNG wire#powerrail
      "Unit1.Em0.StepToString"(StepDINT := "Unit1.Em0.ControlNodes".sepaUnwinderTop.sequence.status.currentStep, Ret_Val => "Unit1.Em0.ControlNodes".sepaUnwinderTop.sequence.status.currentStepSTRING)
   END_RUNG
   RUNG wire#powerrail
      "Unit1.Em0.StepToString"(StepDINT := "Unit1.Em0.ControlNodes".sepaUnwinderTop.sequence.status.previousStep, Ret_Val => "Unit1.Em0.ControlNodes".sepaUnwinderTop.sequence.status.previousStepSTRING)
   END_RUNG
   RUNG wire#powerrail
      "Unit1.Em0.StepToString"(StepDINT := "Unit1.Em0.ControlNodes".sepaUnwinderTop.sequence.status.nextStep, Ret_Val => "Unit1.Em0.ControlNodes".sepaUnwinderTop.sequence.status.nextStepSTRING)
   END_RUNG
   // the same network as SCL:
   "Unit1.Em0.ControlNodes".sepaUnwinderTop.sequence.status.currentStepSTRING := "Unit1.Em0.StepToString"(StepDINT := "Unit1.Em0.ControlNodes".sepaUnwinderTop.sequence.status.currentStep);
   "Unit1.Em0.ControlNodes".sepaUnwinderTop.sequence.status.previousStepSTRING := "Unit1.Em0.StepToString"(StepDINT := "Unit1.Em0.ControlNodes".sepaUnwinderTop.sequence.status.previousStep);
   "Unit1.Em0.ControlNodes".sepaUnwinderTop.sequence.status.nextStepSTRING := "Unit1.Em0.StepToString"(StepDINT := "Unit1.Em0.ControlNodes".sepaUnwinderTop.sequence.status.nextStep);
END_REGION
END_FUNCTION_BLOCK
